PROGRAM MAIN
VAR
	nCounter		: INT;
END_VAR


nCounter	:= nCounter + 1;

END_PROGRAM

(* stored: Version 1.1.0.1, ProductVersion 3.1.4024.4
   POU MAIN: Id {d42d2ce2-876a-4577-ab37-31f0586b6854}, SpecialFunc None *)
